INTERFACE I_AveVoladora

END_INTERFACE

(* stored: Version 1.1.0.1, ProductVersion 3.1.4024.12
   Itf I_AveVoladora: Id {d21195ed-9f61-45e8-b1b1-886005619c2c} *)
